(* Logix 5000 project; controller Amvex_Thorpe_Flowmeter vendor 1 type 14 code 106 rev 33.13; software revision 33.01; part 8 of 16 *)
(* tags used below, declared in another part *)
   Close : BOOL;
   Open : BOOL;
   Torque : DINT;

ADD_ON_INSTRUCTION SetJointVel   (* revision 0.1, vendor Mecademic Inc., ExecuteEnableInFalse *)
// Set joint target velocity in percent (for MovePost and MoveJoint only)
VAR_IN_OUT
   RobotInputs : _061D:Meca500_86BDA20B:I:0; {required}
   RobotOutputs : _061D:Meca500_01F88326:O:0; {required}
END_VAR
VAR_INPUT
   Parameter_Value : REAL; {required}
   ExternalStateControl : BOOL; {required}
   ExternalMoveID : INT; {required}
END_VAR
VAR_OUTPUT
   Enabled : BOOL; {visible}
   Sent : BOOL; {visible}
   Buffered : BOOL; {visible}
   Error : BOOL; {visible}
END_VAR
VAR
   InternalMoveID : INT; {access None}
   MoveIDTrig : BOOL; {access None}
   MoveIDUpdated : BOOL; {access None}
   OneShot : DINT; {access None}
   FirstScan : BOOL; {access None}
END_VAR

ROUTINE EnableInFalse   (* ladder *)
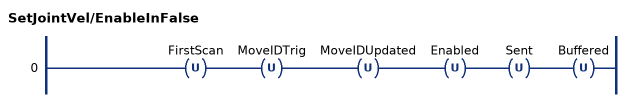
   0: OTU(FirstScan)OTU(MoveIDTrig)OTU(MoveIDUpdated)OTU(Enabled)OTU(Sent)OTU(Buffered);
END_ROUTINE

ROUTINE Logic   (* ladder *)
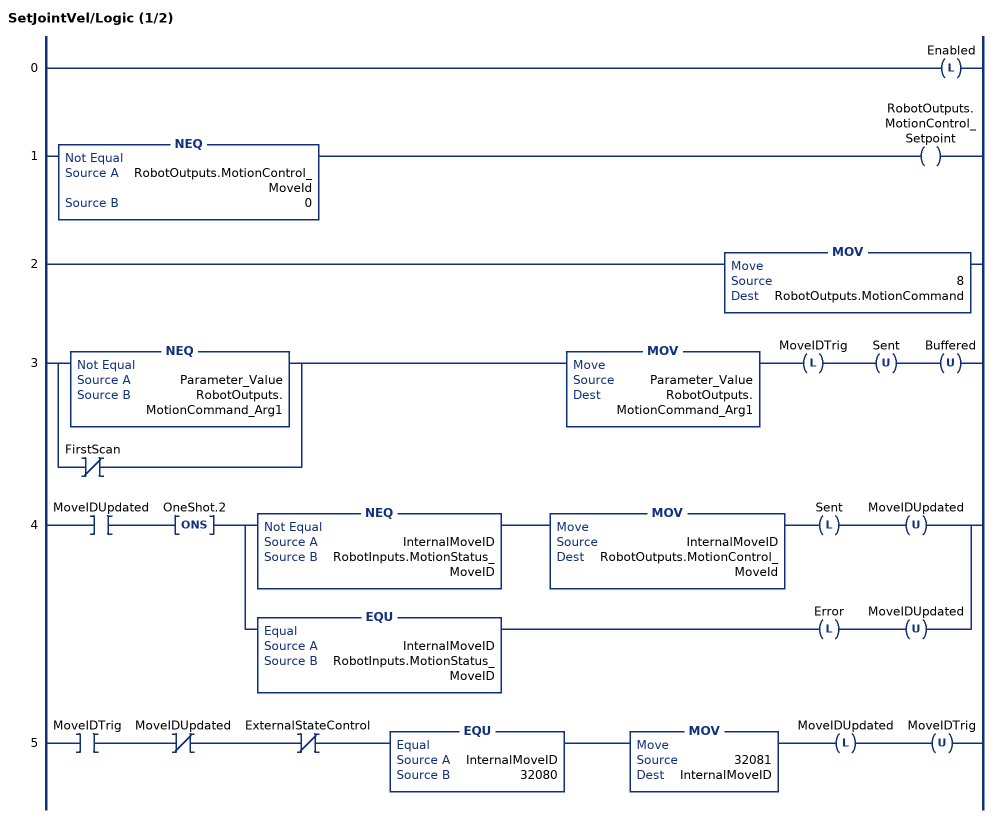
   0: OTL(Enabled);
   1: NEQ(RobotOutputs.MotionControl_MoveId,0)OTE(RobotOutputs.MotionControl_Setpoint);
   2: MOV(8,RobotOutputs.MotionCommand);
   3: [NEQ(Parameter_Value,RobotOutputs.MotionCommand_Arg1) ,XIO(FirstScan) ]MOV(Parameter_Value,RobotOutputs.MotionCommand_Arg1)OTL(MoveIDTrig)OTU(Sent)OTU(Buffered);
   4: XIC(MoveIDUpdated)ONS(OneShot.2)[NEQ(InternalMoveID,RobotInputs.MotionStatus_MoveID) MOV(InternalMoveID,RobotOutputs.MotionControl_MoveId) OTL(Sent) OTU(MoveIDUpdated) ,EQU(InternalMoveID,RobotInputs.MotionStatus_MoveID) OTL(Error) OTU(MoveIDUpdated) ];
   5: XIC(MoveIDTrig)XIO(MoveIDUpdated)XIO(ExternalStateControl)EQU(InternalMoveID,32080)MOV(32081,InternalMoveID)OTL(MoveIDUpdated)OTU(MoveIDTrig);
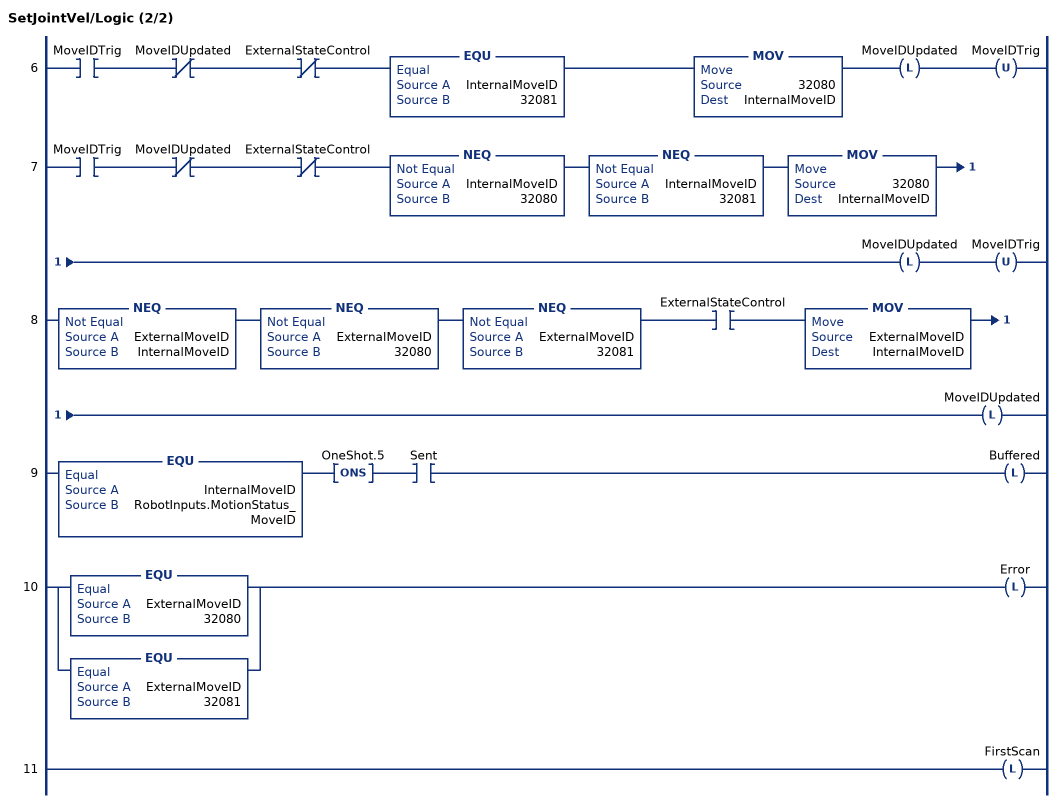
   6: XIC(MoveIDTrig)XIO(MoveIDUpdated)XIO(ExternalStateControl)EQU(InternalMoveID,32081)MOV(32080,InternalMoveID)OTL(MoveIDUpdated)OTU(MoveIDTrig);
   7: XIC(MoveIDTrig)XIO(MoveIDUpdated)XIO(ExternalStateControl)NEQ(InternalMoveID,32080)NEQ(InternalMoveID,32081)MOV(32080,InternalMoveID)OTL(MoveIDUpdated)OTU(MoveIDTrig);
   8: NEQ(ExternalMoveID,InternalMoveID)NEQ(ExternalMoveID,32080)NEQ(ExternalMoveID,32081)XIC(ExternalStateControl)MOV(ExternalMoveID,InternalMoveID)OTL(MoveIDUpdated);
   9: EQU(InternalMoveID,RobotInputs.MotionStatus_MoveID)ONS(OneShot.5)XIC(Sent)OTL(Buffered);
   10: [EQU(ExternalMoveID,32080) ,EQU(ExternalMoveID,32081) ]OTL(Error);
   11: OTL(FirstScan);
END_ROUTINE
END_ADD_ON_INSTRUCTION

ADD_ON_INSTRUCTION SetTorqueLimits   (* revision 0.1, vendor Mecademic Inc., ExecuteEnableInFalse *)
// Set torque limits for current motion
VAR_IN_OUT
   RobotInputs : _061D:Meca500_86BDA20B:I:0; {required}
   RobotOutputs : _061D:Meca500_01F88326:O:0; {required}
END_VAR
VAR_INPUT
   Joint_1_Limit : REAL; {required}
   Joint_2_Limit : REAL; {required}
   Joint_3_Limit : REAL; {required}
   Joint_4_Limit : REAL; {required}
   Joint_5_Limit : REAL; {required}
   Joint_6_Limit : REAL; {required}
   ExternalStateControl : BOOL; {required}
   ExternalMoveID : INT; {required}
END_VAR
VAR_OUTPUT
   Enabled : BOOL; {visible}
   Sent : BOOL; {visible}
   Buffered : BOOL; {visible}
   Error : BOOL; {visible}
END_VAR
VAR
   InternalMoveID : INT; {access None}
   MoveIDUpdated : BOOL; {access None}
   OneShot : DINT; {access None}
   MoveIDTrig : BOOL; {access None}
   FirstScan : BOOL; {access None}
END_VAR

ROUTINE EnableInFalse   (* ladder *)
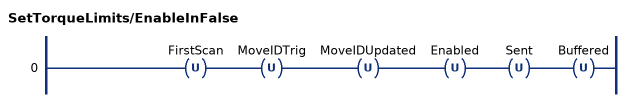
   0: OTU(FirstScan)OTU(MoveIDTrig)OTU(MoveIDUpdated)OTU(Enabled)OTU(Sent)OTU(Buffered);
END_ROUTINE

ROUTINE Logic   (* ladder *)
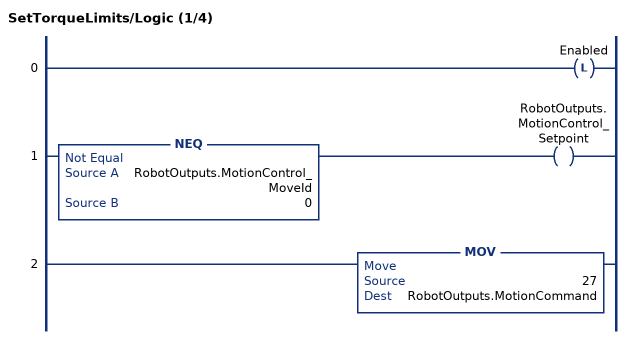
   0: OTL(Enabled);
   1: NEQ(RobotOutputs.MotionControl_MoveId,0)OTE(RobotOutputs.MotionControl_Setpoint);
   2: MOV(27,RobotOutputs.MotionCommand);
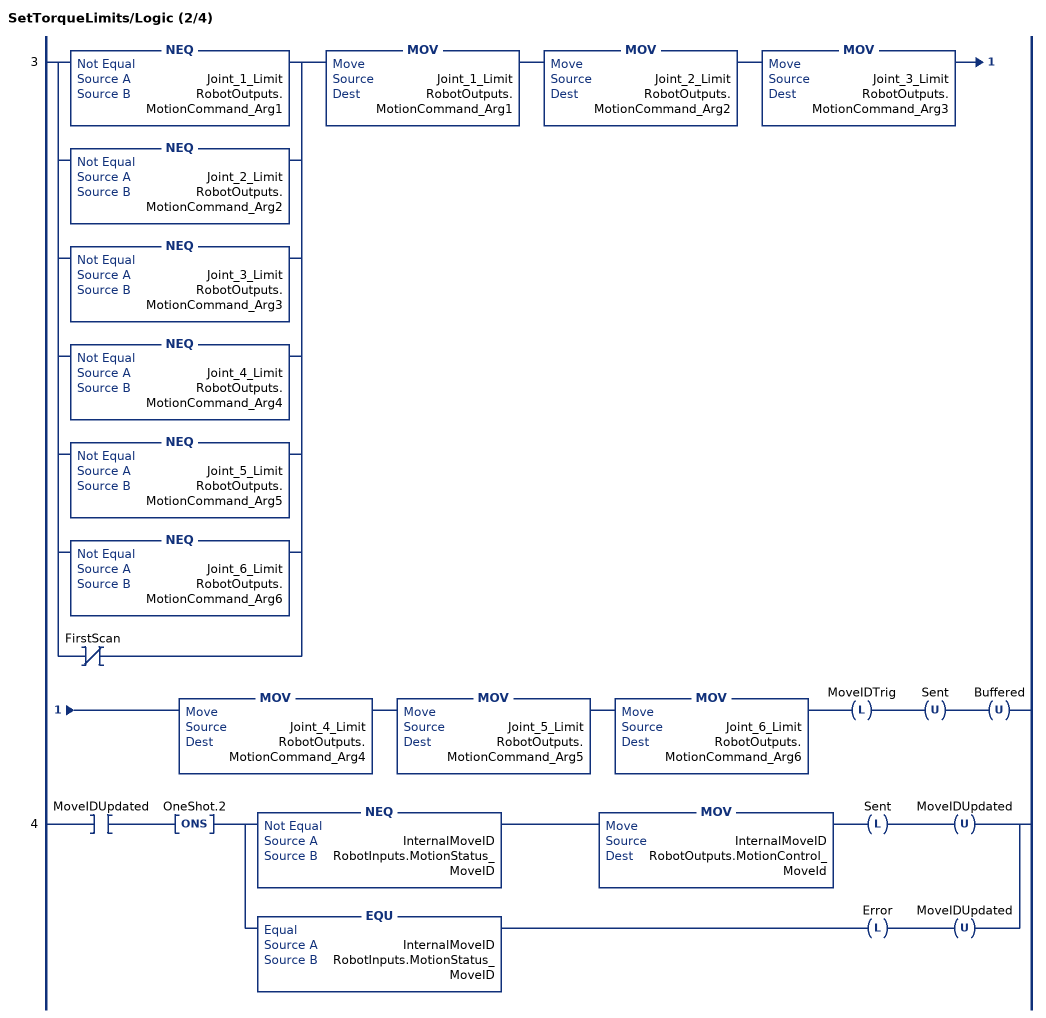
   3: [NEQ(Joint_1_Limit,RobotOutputs.MotionCommand_Arg1) ,NEQ(Joint_2_Limit,RobotOutputs.MotionCommand_Arg2) ,NEQ(Joint_3_Limit,RobotOutputs.MotionCommand_Arg3) ,NEQ(Joint_4_Limit,RobotOutputs.MotionCommand_Arg4) ,NEQ(Joint_5_Limit,RobotOutputs.MotionCommand_Arg5) ,NEQ(Joint_6_Limit,RobotOutputs.MotionCommand_Arg6) ,XIO(FirstScan) ]MOV(Joint_1_Limit,RobotOutputs.MotionCommand_Arg1)MOV(Joint_2_Limit,RobotOutputs.MotionCommand_Arg2)MOV(Joint_3_Limit,RobotOutputs.MotionCommand_Arg3)MOV(Joint_4_Limit,RobotOutputs.MotionCommand_Arg4)MOV(Joint_5_Limit,RobotOutputs.MotionCommand_Arg5)MOV(Joint_6_Limit,RobotOutputs.MotionCommand_Arg6)OTL(MoveIDTrig)OTU(Sent)OTU(Buffered);
   4: XIC(MoveIDUpdated)ONS(OneShot.2)[NEQ(InternalMoveID,RobotInputs.MotionStatus_MoveID) MOV(InternalMoveID,RobotOutputs.MotionControl_MoveId) OTL(Sent) OTU(MoveIDUpdated) ,EQU(InternalMoveID,RobotInputs.MotionStatus_MoveID) OTL(Error) OTU(MoveIDUpdated) ];
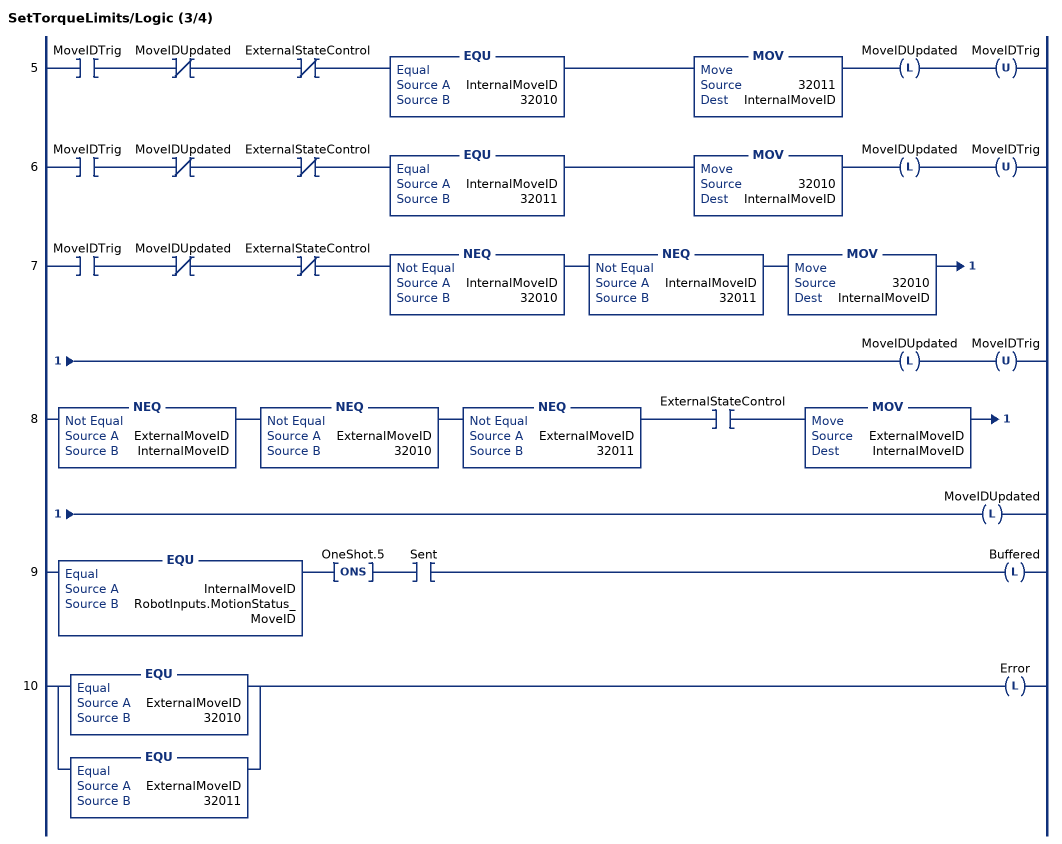
   5: XIC(MoveIDTrig)XIO(MoveIDUpdated)XIO(ExternalStateControl)EQU(InternalMoveID,32010)MOV(32011,InternalMoveID)OTL(MoveIDUpdated)OTU(MoveIDTrig);
   6: XIC(MoveIDTrig)XIO(MoveIDUpdated)XIO(ExternalStateControl)EQU(InternalMoveID,32011)MOV(32010,InternalMoveID)OTL(MoveIDUpdated)OTU(MoveIDTrig);
   7: XIC(MoveIDTrig)XIO(MoveIDUpdated)XIO(ExternalStateControl)NEQ(InternalMoveID,32010)NEQ(InternalMoveID,32011)MOV(32010,InternalMoveID)OTL(MoveIDUpdated)OTU(MoveIDTrig);
   8: NEQ(ExternalMoveID,InternalMoveID)NEQ(ExternalMoveID,32010)NEQ(ExternalMoveID,32011)XIC(ExternalStateControl)MOV(ExternalMoveID,InternalMoveID)OTL(MoveIDUpdated);
   9: EQU(InternalMoveID,RobotInputs.MotionStatus_MoveID)ONS(OneShot.5)XIC(Sent)OTL(Buffered);
   10: [EQU(ExternalMoveID,32010) ,EQU(ExternalMoveID,32011) ]OTL(Error);
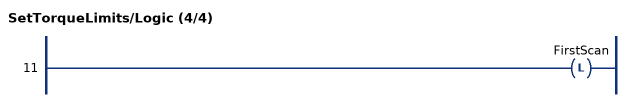
   11: OTL(FirstScan);
END_ROUTINE
END_ADD_ON_INSTRUCTION

ADD_ON_INSTRUCTION SetTorqueLimitsCfg   (* revision 0.1, vendor Mecademic Inc., ExecuteEnableInFalse *)
// Enable torque limits for current motion
VAR_IN_OUT
   RobotInputs : _061D:Meca500_86BDA20B:I:0; {required}
   RobotOutputs : _061D:Meca500_01F88326:O:0; {required}
END_VAR
VAR_INPUT
   Severity : REAL; {required}
   Detection_Mode : REAL; {required}
   ExternalStateControl : BOOL; {required}
   ExternalMoveID : INT; {required}
END_VAR
VAR_OUTPUT
   Enabled : BOOL; {visible}
   Sent : BOOL; {visible}
   Buffered : BOOL; {visible}
   Error : BOOL; {visible}
END_VAR
VAR
   InternalMoveID : INT; {access None}
   MoveIDUpdated : BOOL; {access None}
   OneShot : DINT; {access None}
   MoveIDTrig : BOOL; {access None}
   FirstScan : BOOL; {access None}
END_VAR

ROUTINE EnableInFalse   (* ladder *)
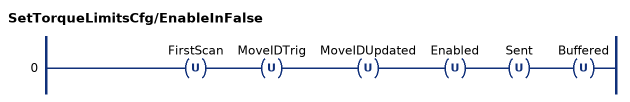
   0: OTU(FirstScan)OTU(MoveIDTrig)OTU(MoveIDUpdated)OTU(Enabled)OTU(Sent)OTU(Buffered);
END_ROUTINE

ROUTINE Logic   (* ladder *)
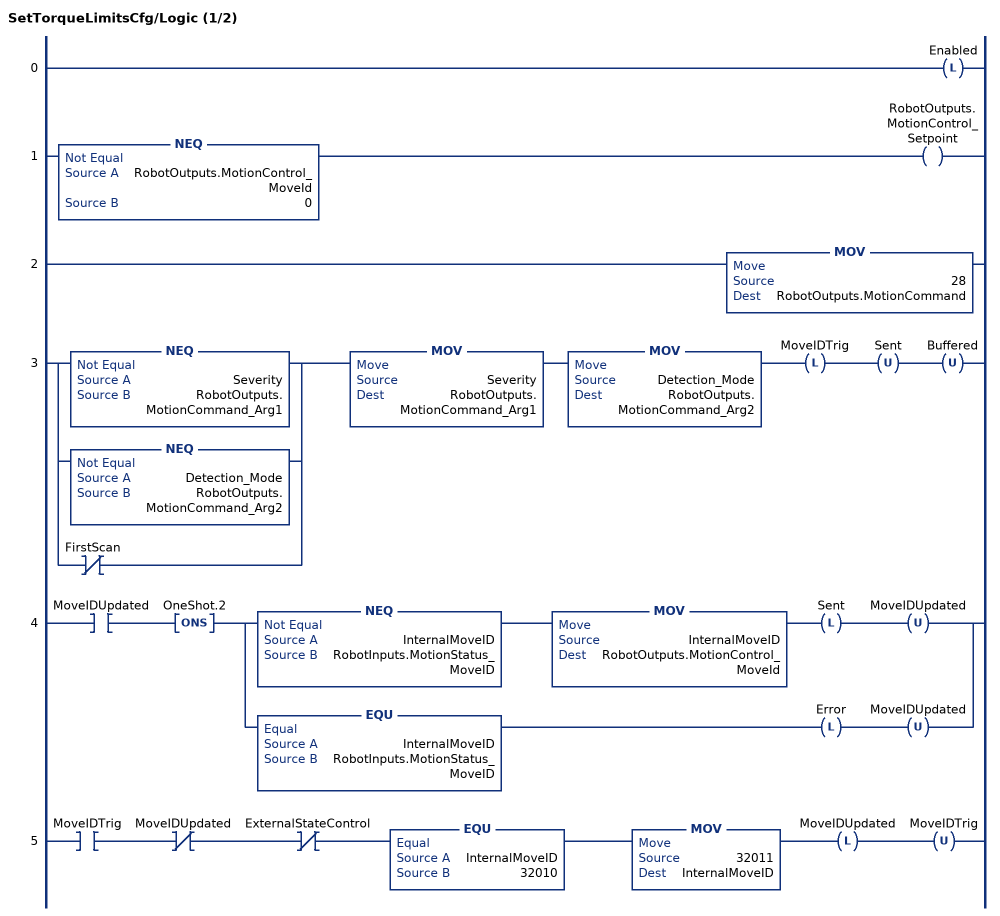
   0: OTL(Enabled);
   1: NEQ(RobotOutputs.MotionControl_MoveId,0)OTE(RobotOutputs.MotionControl_Setpoint);
   2: MOV(28,RobotOutputs.MotionCommand);
   3: [NEQ(Severity,RobotOutputs.MotionCommand_Arg1) ,NEQ(Detection_Mode,RobotOutputs.MotionCommand_Arg2) ,XIO(FirstScan) ]MOV(Severity,RobotOutputs.MotionCommand_Arg1)MOV(Detection_Mode,RobotOutputs.MotionCommand_Arg2)OTL(MoveIDTrig)OTU(Sent)OTU(Buffered);
   4: XIC(MoveIDUpdated)ONS(OneShot.2)[NEQ(InternalMoveID,RobotInputs.MotionStatus_MoveID) MOV(InternalMoveID,RobotOutputs.MotionControl_MoveId) OTL(Sent) OTU(MoveIDUpdated) ,EQU(InternalMoveID,RobotInputs.MotionStatus_MoveID) OTL(Error) OTU(MoveIDUpdated) ];
   5: XIC(MoveIDTrig)XIO(MoveIDUpdated)XIO(ExternalStateControl)EQU(InternalMoveID,32010)MOV(32011,InternalMoveID)OTL(MoveIDUpdated)OTU(MoveIDTrig);
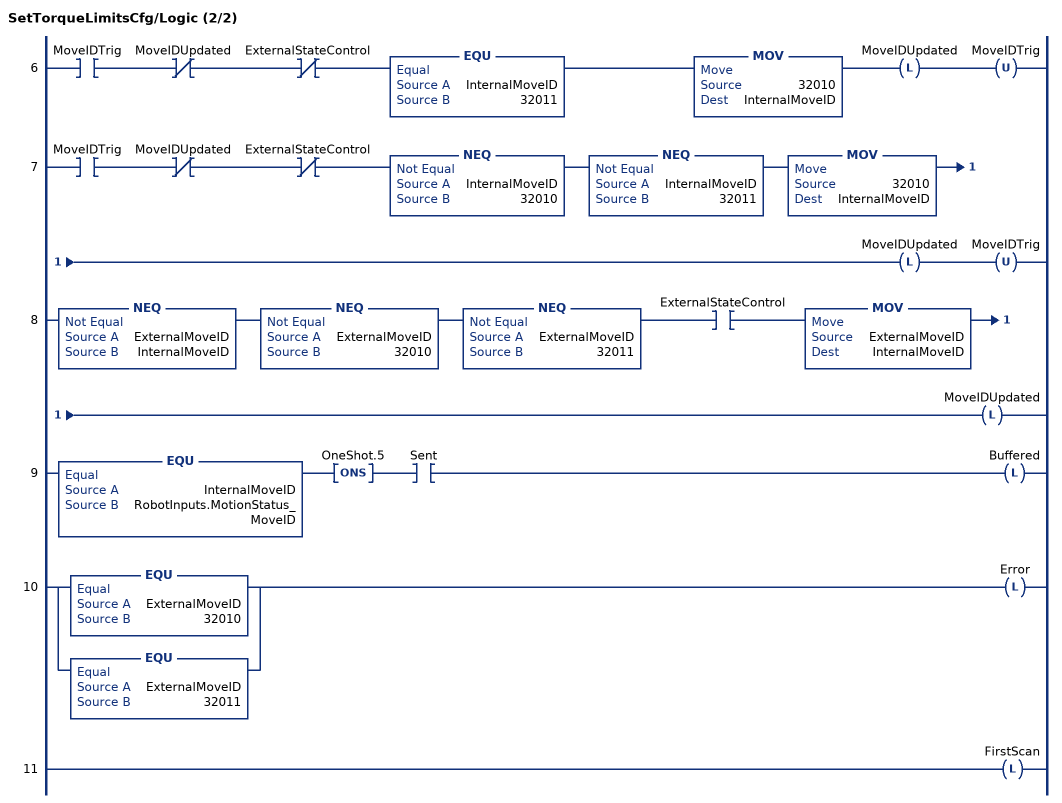
   6: XIC(MoveIDTrig)XIO(MoveIDUpdated)XIO(ExternalStateControl)EQU(InternalMoveID,32011)MOV(32010,InternalMoveID)OTL(MoveIDUpdated)OTU(MoveIDTrig);
   7: XIC(MoveIDTrig)XIO(MoveIDUpdated)XIO(ExternalStateControl)NEQ(InternalMoveID,32010)NEQ(InternalMoveID,32011)MOV(32010,InternalMoveID)OTL(MoveIDUpdated)OTU(MoveIDTrig);
   8: NEQ(ExternalMoveID,InternalMoveID)NEQ(ExternalMoveID,32010)NEQ(ExternalMoveID,32011)XIC(ExternalStateControl)MOV(ExternalMoveID,InternalMoveID)OTL(MoveIDUpdated);
   9: EQU(InternalMoveID,RobotInputs.MotionStatus_MoveID)ONS(OneShot.5)XIC(Sent)OTL(Buffered);
   10: [EQU(ExternalMoveID,32010) ,EQU(ExternalMoveID,32011) ]OTL(Error);
   11: OTL(FirstScan);
END_ROUTINE
END_ADD_ON_INSTRUCTION

ADD_ON_INSTRUCTION SetTRF   (* revision 0.1, vendor Mecademic Inc., ExecuteEnableInFalse *)
// Set the pose of the RTF with respect of the FRF
VAR_IN_OUT
   RobotInputs : _061D:Meca500_86BDA20B:I:0; {required}
   RobotOutputs : _061D:Meca500_01F88326:O:0; {required}
END_VAR
VAR_INPUT
   Pose_X_Pos : REAL; {required}
   Pose_Y_Pos : REAL; {required}
   Pose_Z_Pos : REAL; {required}
   Pose_rX_Ang : REAL; {required}
   Pose_rY_Ang : REAL; {required}
   Pose_rZ_Ang : REAL; {required}
   ExternalStateControl : BOOL; {required}
   ExternalMoveID : INT; {required}
END_VAR
VAR_OUTPUT
   Enabled : BOOL; {visible}
   Sent : BOOL; {visible}
   Buffered : BOOL; {visible}
   Error : BOOL; {visible}
END_VAR
VAR
   InternalMoveID : INT; {access None}
   MoveIDTrig : BOOL; {access None}
   MoveIDUpdated : BOOL; {access None}
   OneShot : DINT; {access None}
   FirstScan : BOOL; {access None}
END_VAR

ROUTINE EnableInFalse   (* ladder *)
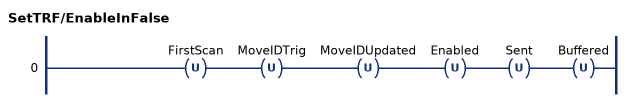
   0: OTU(FirstScan)OTU(MoveIDTrig)OTU(MoveIDUpdated)OTU(Enabled)OTU(Sent)OTU(Buffered);
END_ROUTINE

ROUTINE Logic   (* ladder *)
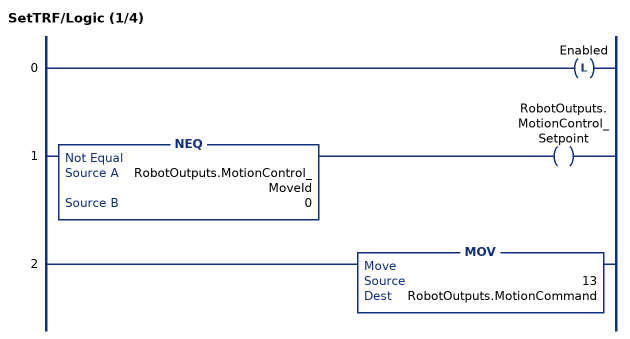
   0: OTL(Enabled);
   1: NEQ(RobotOutputs.MotionControl_MoveId,0)OTE(RobotOutputs.MotionControl_Setpoint);
   2: MOV(13,RobotOutputs.MotionCommand);
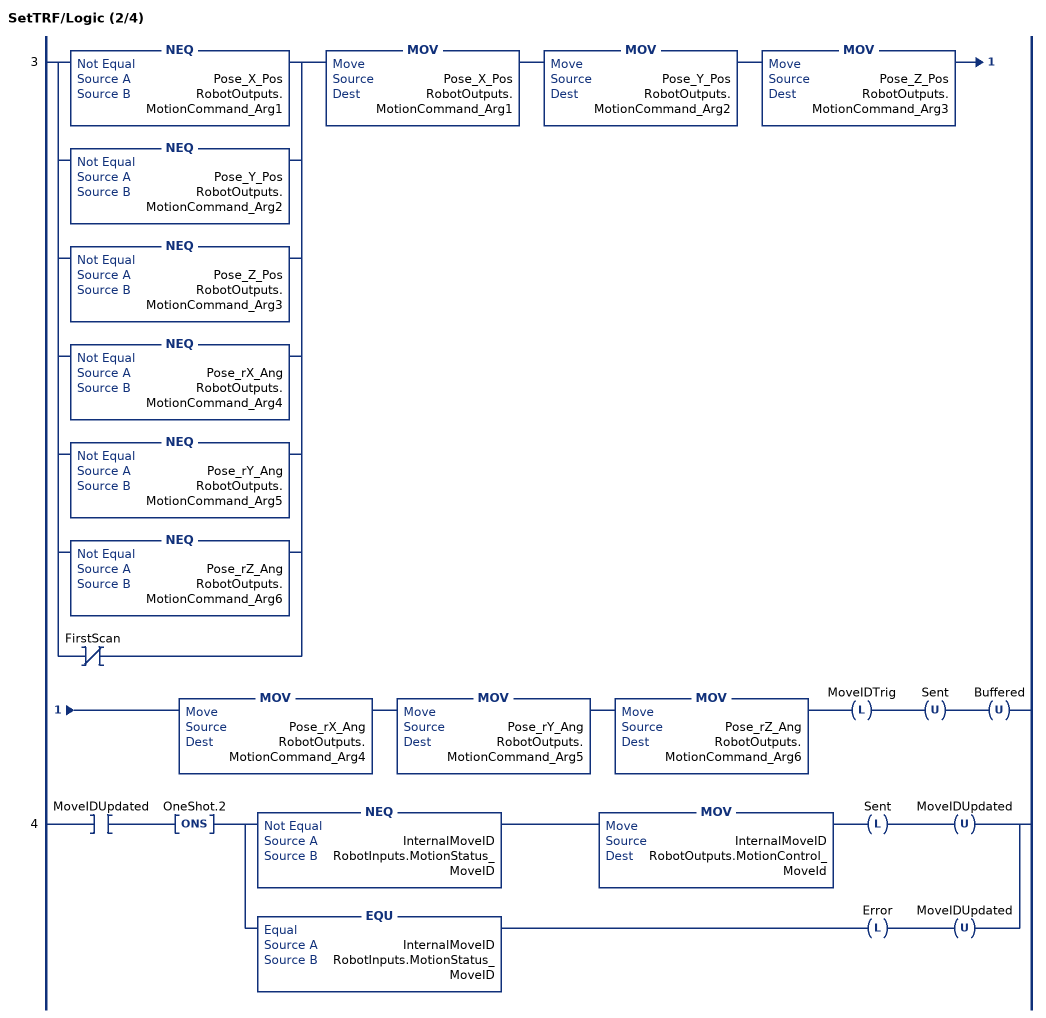
   3: [NEQ(Pose_X_Pos,RobotOutputs.MotionCommand_Arg1) ,NEQ(Pose_Y_Pos,RobotOutputs.MotionCommand_Arg2) ,NEQ(Pose_Z_Pos,RobotOutputs.MotionCommand_Arg3) ,NEQ(Pose_rX_Ang,RobotOutputs.MotionCommand_Arg4) ,NEQ(Pose_rY_Ang,RobotOutputs.MotionCommand_Arg5) ,NEQ(Pose_rZ_Ang,RobotOutputs.MotionCommand_Arg6) ,XIO(FirstScan) ]MOV(Pose_X_Pos,RobotOutputs.MotionCommand_Arg1)MOV(Pose_Y_Pos,RobotOutputs.MotionCommand_Arg2)MOV(Pose_Z_Pos,RobotOutputs.MotionCommand_Arg3)MOV(Pose_rX_Ang,RobotOutputs.MotionCommand_Arg4)MOV(Pose_rY_Ang,RobotOutputs.MotionCommand_Arg5)MOV(Pose_rZ_Ang,RobotOutputs.MotionCommand_Arg6)OTL(MoveIDTrig)OTU(Sent)OTU(Buffered);
   4: XIC(MoveIDUpdated)ONS(OneShot.2)[NEQ(InternalMoveID,RobotInputs.MotionStatus_MoveID) MOV(InternalMoveID,RobotOutputs.MotionControl_MoveId) OTL(Sent) OTU(MoveIDUpdated) ,EQU(InternalMoveID,RobotInputs.MotionStatus_MoveID) OTL(Error) OTU(MoveIDUpdated) ];
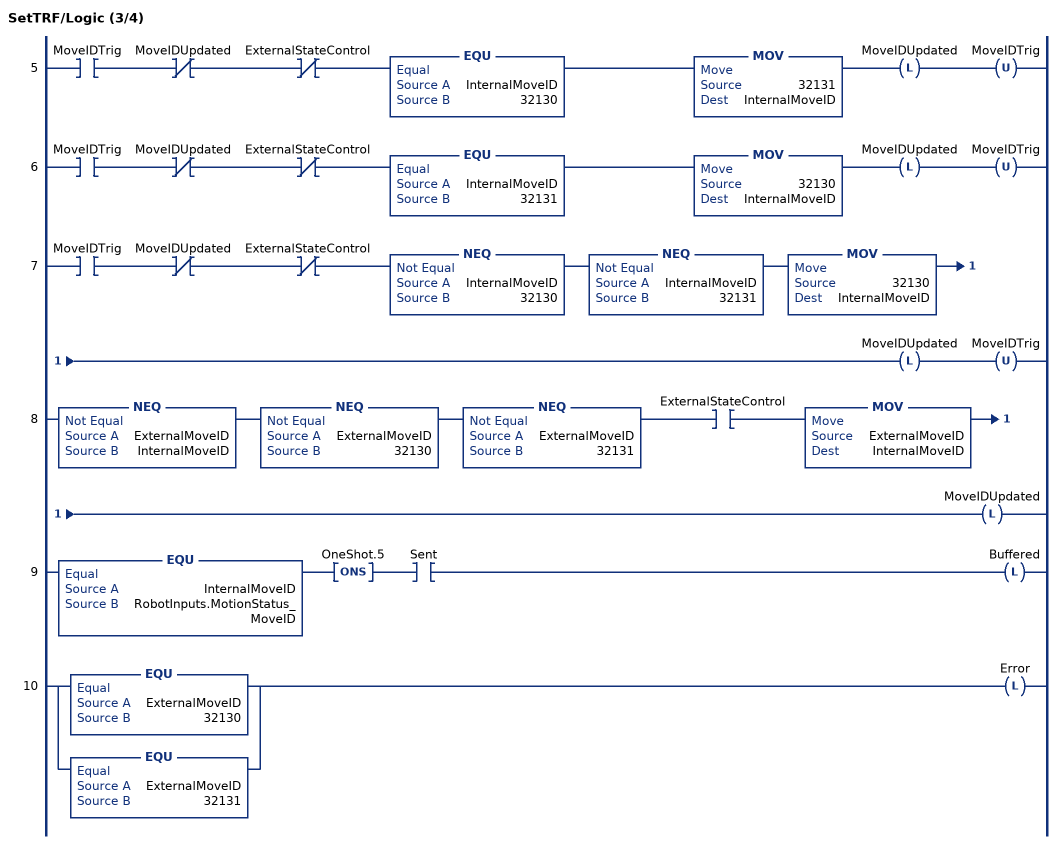
   5: XIC(MoveIDTrig)XIO(MoveIDUpdated)XIO(ExternalStateControl)EQU(InternalMoveID,32130)MOV(32131,InternalMoveID)OTL(MoveIDUpdated)OTU(MoveIDTrig);
   6: XIC(MoveIDTrig)XIO(MoveIDUpdated)XIO(ExternalStateControl)EQU(InternalMoveID,32131)MOV(32130,InternalMoveID)OTL(MoveIDUpdated)OTU(MoveIDTrig);
   7: XIC(MoveIDTrig)XIO(MoveIDUpdated)XIO(ExternalStateControl)NEQ(InternalMoveID,32130)NEQ(InternalMoveID,32131)MOV(32130,InternalMoveID)OTL(MoveIDUpdated)OTU(MoveIDTrig);
   8: NEQ(ExternalMoveID,InternalMoveID)NEQ(ExternalMoveID,32130)NEQ(ExternalMoveID,32131)XIC(ExternalStateControl)MOV(ExternalMoveID,InternalMoveID)OTL(MoveIDUpdated);
   9: EQU(InternalMoveID,RobotInputs.MotionStatus_MoveID)ONS(OneShot.5)XIC(Sent)OTL(Buffered);
   10: [EQU(ExternalMoveID,32130) ,EQU(ExternalMoveID,32131) ]OTL(Error);
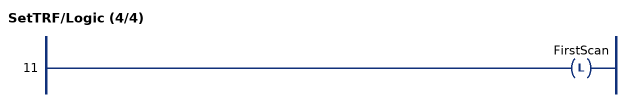
   11: OTL(FirstScan);
END_ROUTINE
END_ADD_ON_INSTRUCTION

ADD_ON_INSTRUCTION SetValveState   (* revision 1.0, vendor Mecademic inc., ExecuteEnableInFalse *)
// Set valve box states (0.close, 1.open, -1.stay)
VAR_OUTPUT
   Enabled : BOOL; {access Read Only, visible}
END_VAR
VAR_IN_OUT
   RobotOutputs : _061D:Meca500_01F88326:O:0; {required}
   RobotInputs : _061D:Meca500_86BDA20B:I:0; {required}
END_VAR
VAR_INPUT
   Valve_1_State : DINT; {required}   // -1 = Close, 0 = Stay, 1 = Open
   Valve_2_State : DINT; {required}   // -1 = Close, 0 = Stay, 1 = Open
END_VAR
VAR_OUTPUT
   Sent : BOOL; {access Read Only, visible}
   Buffered : BOOL; {access Read Only, visible}
   Error : BOOL; {access Read Only, visible}
END_VAR
VAR_INPUT
   ExternalStateControl : BOOL; {required}
   ExternalMoveID : INT; {required}
END_VAR
VAR
   MoveIDTrig : BOOL; {access None}
   FirstScan : BOOL; {access None}
   MoveIDUpdated : BOOL; {access None}
   OneShot : DINT; {access None}
   InternalMoveID : DINT; {access None}
END_VAR

ROUTINE EnableInFalse   (* ladder *)
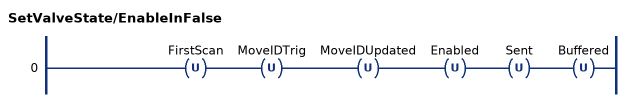
   0: OTU(FirstScan)OTU(MoveIDTrig)OTU(MoveIDUpdated)OTU(Enabled)OTU(Sent)OTU(Buffered);
END_ROUTINE

ROUTINE Logic   (* ladder *)
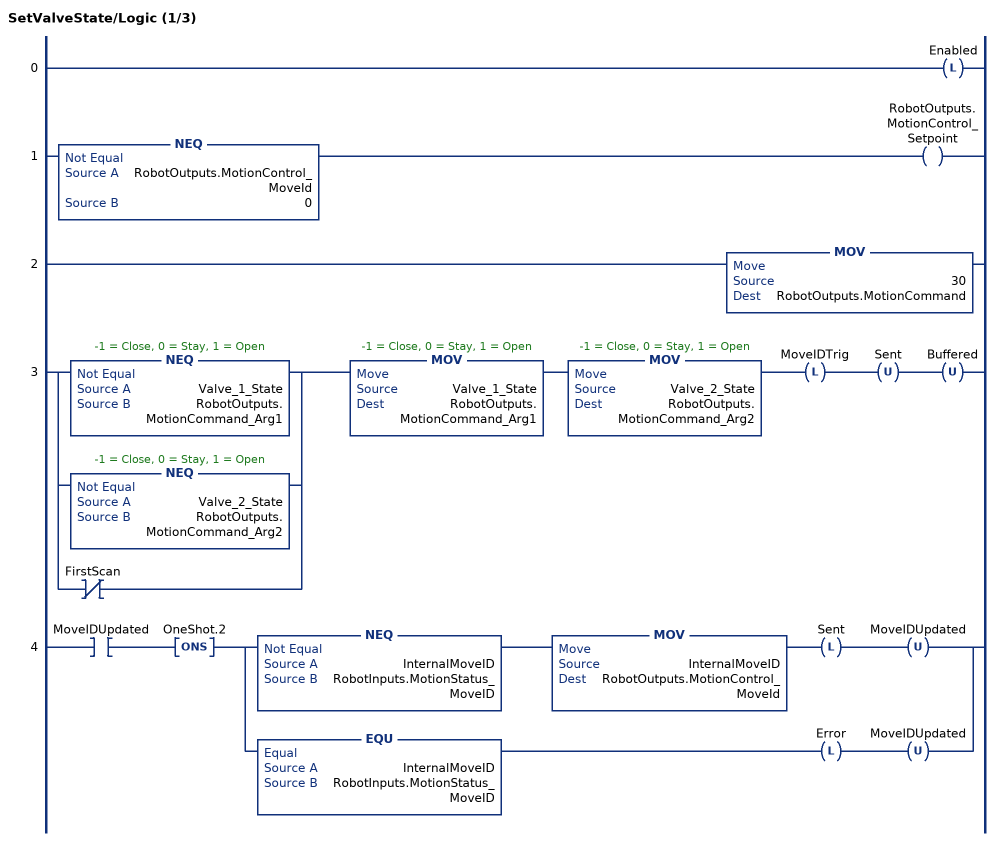
   0: OTL(Enabled);
   1: NEQ(RobotOutputs.MotionControl_MoveId,0)OTE(RobotOutputs.MotionControl_Setpoint);
   2: MOV(30,RobotOutputs.MotionCommand);
   3: [NEQ(Valve_1_State,RobotOutputs.MotionCommand_Arg1) ,NEQ(Valve_2_State,RobotOutputs.MotionCommand_Arg2) ,XIO(FirstScan) ]MOV(Valve_1_State,RobotOutputs.MotionCommand_Arg1)MOV(Valve_2_State,RobotOutputs.MotionCommand_Arg2)OTL(MoveIDTrig)OTU(Sent)OTU(Buffered);
   4: XIC(MoveIDUpdated)ONS(OneShot.2)[NEQ(InternalMoveID,RobotInputs.MotionStatus_MoveID) MOV(InternalMoveID,RobotOutputs.MotionControl_MoveId) OTL(Sent) OTU(MoveIDUpdated) ,EQU(InternalMoveID,RobotInputs.MotionStatus_MoveID) OTL(Error) OTU(MoveIDUpdated) ];
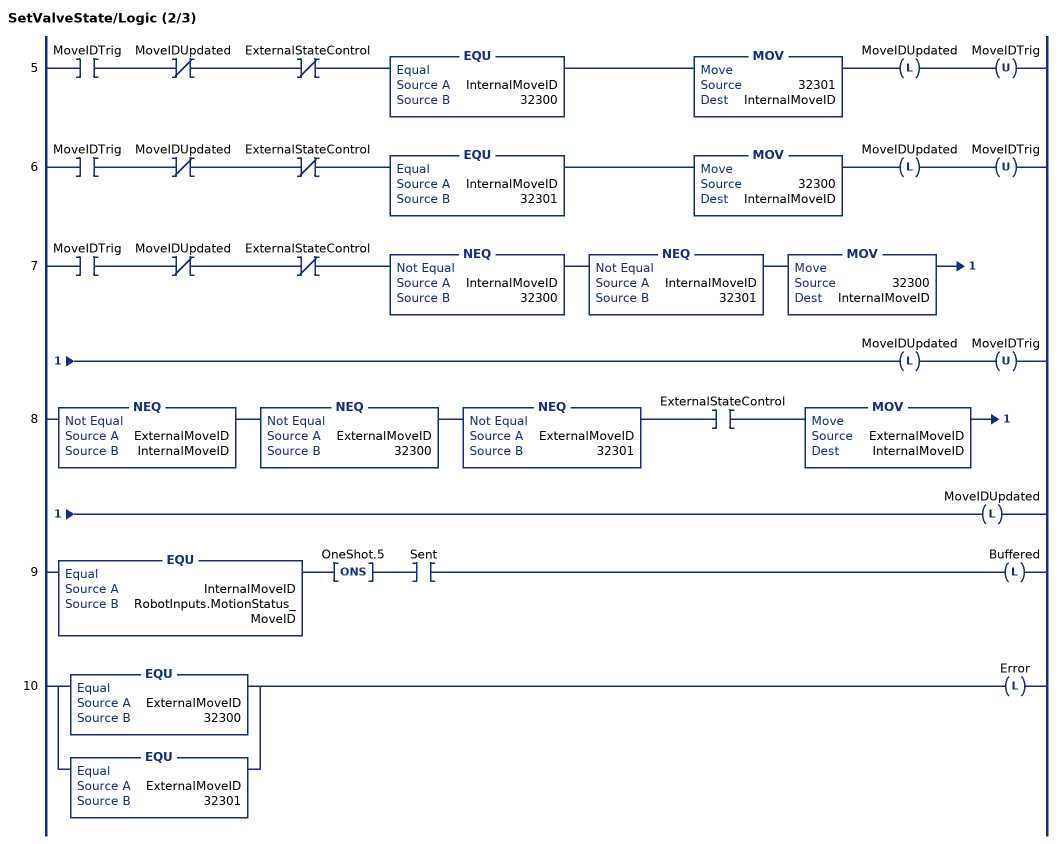
   5: XIC(MoveIDTrig)XIO(MoveIDUpdated)XIO(ExternalStateControl)EQU(InternalMoveID,32300)MOV(32301,InternalMoveID)OTL(MoveIDUpdated)OTU(MoveIDTrig);
   6: XIC(MoveIDTrig)XIO(MoveIDUpdated)XIO(ExternalStateControl)EQU(InternalMoveID,32301)MOV(32300,InternalMoveID)OTL(MoveIDUpdated)OTU(MoveIDTrig);
   7: XIC(MoveIDTrig)XIO(MoveIDUpdated)XIO(ExternalStateControl)NEQ(InternalMoveID,32300)NEQ(InternalMoveID,32301)MOV(32300,InternalMoveID)OTL(MoveIDUpdated)OTU(MoveIDTrig);
   8: NEQ(ExternalMoveID,InternalMoveID)NEQ(ExternalMoveID,32300)NEQ(ExternalMoveID,32301)XIC(ExternalStateControl)MOV(ExternalMoveID,InternalMoveID)OTL(MoveIDUpdated);
   9: EQU(InternalMoveID,RobotInputs.MotionStatus_MoveID)ONS(OneShot.5)XIC(Sent)OTL(Buffered);
   10: [EQU(ExternalMoveID,32300) ,EQU(ExternalMoveID,32301) ]OTL(Error);
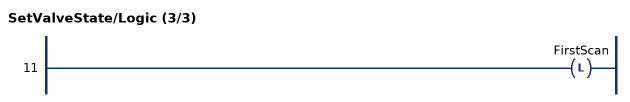
   11: OTL(FirstScan);
END_ROUTINE
END_ADD_ON_INSTRUCTION
